PROGRAM MAIN
VAR
	fbEvent:		FB_Event;
	fbHandler:		FB_Events;
	bInit:			BOOL:= TRUE;;
	bEvent: 		BOOL;
END_VAR

IF bInit THEN
	bInit:= FALSE;
	fbEvent.P_Handler:= fbHandler;
END_IF

fbHandler();

IF bEvent THEN
	fbEvent.M_Critical(E_Type.Error, 'Message', 1);
END_IF

END_PROGRAM

(* stored: Version 1.1.0.1, ProductVersion 3.1.4024.12
   POU MAIN: Id {e5f7a5a1-3f48-4670-a47b-5f2ccf40d0d9}, SpecialFunc None *)
